FUNCTION_BLOCK FB_AxisHardware
VAR_INPUT
	bExecute: BOOL;
	amsEncAddr: AMSADDR;
	nEncCh: USINT;
END_VAR
VAR_IN_OUT
	Axis: AXIS_REF;
END_VAR
VAR_OUTPUT
	bDone: BOOL;
	bBusy: BOOL;
	bError: BOOL;
	nErrorID: UDINT;
	stHardware: ST_AxisHardware;
END_VAR
VAR
	fbReadDriveAddress: MC_ReadDriveAddress;
	fbDriveId: FB_EcGetSlaveIdentity;
	fbEncId: FB_EcGetSlaveIdentity;
	fbADSRead: ADSREADEX;
	stDriveAddr: ST_DriveAddress;
	stDriveRef: ST_DriveRef;
	stEncRef: ST_DriveRef;
END_VAR

// Get drive ref using AXIS_REF
fbReadDriveAddress(Execute:=bExecute,
	Axis:=Axis,
	DriveAddress=>stDriveAddr);
stDriveRef.sNetId := stDriveAddr.NetID;
stDriveRef.nSlaveAddr := stDriveAddr.SlaveAddress;
stDriveRef.nDriveNo := stDriveAddr.Channel;
stHardware.drive_ref := stDriveRef;

// Get encoder ref using input args (cannot be derived from AXIS_REF)
stEncRef.sNetId := F_CreateAmsNetId(amsEncAddr.netId);
stEncRef.nSlaveAddr := amsEncAddr.port;
stEncRef.nDriveNo := nEncCh;
stHardware.enc_ref := stEncRef;

// Get the drive model (e.g. 7031)
IF stDriveRef.nSlaveAddr > 0 THEN
	fbDriveId(bExecute:=bExecute AND fbReadDriveAddress.Done,
		sNetId:=stDriveRef.sNetId,
		nSlaveAddr:=stDriveRef.nSlaveAddr);
	stHardware.drive_type := UDINT_TO_UINT(SHR(fbDriveID.identity.productCode, 16));
END_IF

// Get the encoder model (e.g. 5042)
IF stEncRef.nSlaveAddr > 0 THEN
	fbEncId(bExecute:=bExecute AND fbReadDriveAddress.Done,
		sNetId:=stEncRef.sNetId,
		nSlaveAddr:=stEncRef.nSlaveAddr);
	stHardware.enc_type := UDINT_TO_UINT(SHR(fbEncID.identity.productCode, 16));
END_IF

// Summarize outputs
bDone := fbReadDriveAddress.Done AND NOT fbDriveId.bBusy AND NOT fbEncId.bBusy;
bBusy := fbReadDriveAddress.Busy OR fbDriveId.bBusy OR fbEncId.bBusy;
bError := fbReadDriveAddress.Error OR fbDriveId.bError OR fbEncId.bError;
IF fbReadDriveAddress.ErrorID > 0 THEN
	nErrorID := fbReadDriveAddress.ErrorID;
ELSIF fbDriveId.nErrId >0 THEN
	nErrorID := fbDriveId.nErrId;
ELSE
	nErrorID := fbEncId.nErrId;
END_IF

END_FUNCTION_BLOCK

(* stored: Version 1.1.0.1, ProductVersion 3.1.4020.14
   POU FB_AxisHardware: Id {1564163d-e493-4d9a-b680-85c98f09b3c4}, SpecialFunc None *)
